FUNCTION_BLOCK FB_Impulse_LongPress
VAR_INPUT
	bInput			:	BOOL;	//Input Schalter oder Taster
	tHigh			:	TIME;						//Zeit (ms) für High
	tLongPress		:	TIME;							
END_VAR
VAR_OUTPUT
	bOut			:	BOOL;
	bOutLong		:	BOOL;
END_VAR
VAR_IN_OUT
	bInputHA		:	BOOL;
END_VAR
VAR CONSTANT
END_VAR
VAR
	fbFtrig			:	F_TRIG;
	bTrigger		:	BOOL;
	bOutTrig		:	BOOL;
	
	tpPulse			:	TP;
	tonLongPress	:	TON;
	
END_VAR
VAR_TEMP

END_VAR


tpPulse		 (IN := bOutTrig, PT := tHigh);
tonLongPress (IN := bInput, PT := tLongPress);

bTrigger 	:= FALSE;
		
fbFtrig(CLK:= bInput, Q=> );

//Normale Tastendruck
bTrigger := bTrigger OR fbFtrig.Q;

//Signal über HA
bTrigger := bTrigger OR bInputHA;

//Wenn normaler Tastendruck und Impuls noch nicht abgelaufen
IF (tpPulse.Q AND NOT bInput) OR bTrigger THEN
	bOut 		:= TRUE;
	bInputHA	:= FALSE;
//Wenn langer Tastendruck
ELSIF tonLongPress.Q OR (tpPulse.Q AND bInput) THEN
	bOutLong	:= TRUE;

//Wenn nichts
ELSE
	bOut 		:= FALSE;
	bOutLong	:= FALSE;
	bInputHA	:= FALSE;
	
	bOutTrig	:= FALSE;
END_IF
	
bOutTrig := bOut OR bOutLong;

END_FUNCTION_BLOCK

(* stored: Version 1.1.0.1, ProductVersion 3.1.4024.4
   POU FB_Impulse_LongPress: Id {3f67f426-ae59-43bf-aa2c-054cccab7491}, SpecialFunc None *)
